% RSLogix 500 project MM2.RSS, saved by version 8.10.00.30 %
PROJECT "UNTITLED"    % processor: Bul.1763 MicroLogix 1100 Series B %

PROGRAM FILES
  LAD 2   4 rungs
  LAD 3 "WATCHDOG"  8 rungs
  LAD 4 "PRODUCT"  8 rungs  % Changes the productcode %

DATA FILES
  O0 OUTPUT  4 elements
  I1 INPUT  6 elements
  S2 STATUS  66 elements
  B3 BINARY  1 elements
  T4 TIMER  3 elements
  C5 COUNTER  1 elements
  R6 CONTROL  1 elements
  N7 INTEGER  3 elements
  F8 FLOAT  100 elements
  ST9   10 elements
  MG13   1 elements
  RIX15   1 elements
  RI16   1 elements

LADDER 2
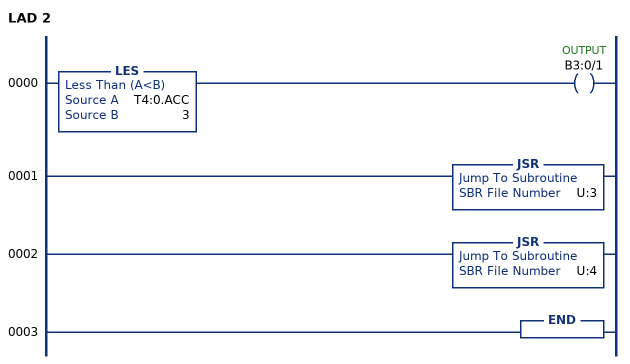
% Rung: 0 %
SOR LES T4:0.ACC 3 OTE B3:0/1 EOR
%   B3:0/1  OUTPUT %
% Rung: 1 %
SOR JSR U:3 EOR
% Rung: 2 %
SOR JSR U:4 EOR
% Rung: 3 %
SOR END EOR

LADDER 3 "WATCHDOG"
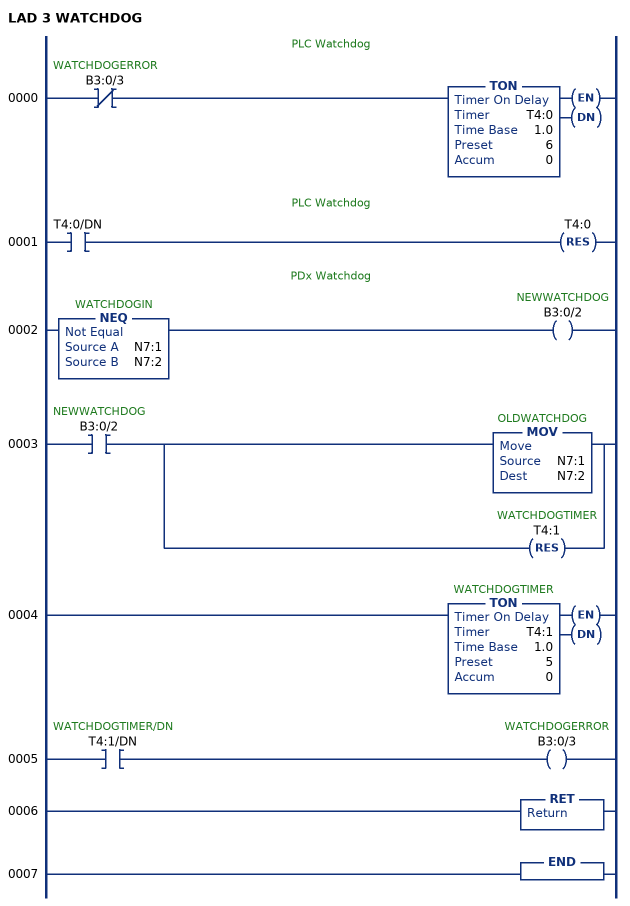
% Rung: 0 %  % edit flag set %
% PLC Watchdog %
SOR XIO B3:0/3 TON T4:0 1.0 6 0 EOR
%   B3:0/3  WATCHDOGERROR %
% Rung: 1 %  % edit flag set %
% PLC Watchdog %
SOR XIC T4:0/DN RES T4:0 EOR
% Rung: 2 %
% PDx Watchdog %
SOR NEQ N7:1 N7:2 OTE B3:0/2 EOR
%   N7:1  WATCHDOGIN %
%   N7:2  OLDWATCHDOG %
%   B3:0/2  NEWWATCHDOG %
% Rung: 3 %
SOR XIC B3:0/2 BST MOV N7:1 N7:2 NXB RES T4:1 BND EOR
%   B3:0/2  NEWWATCHDOG %
%   N7:1  WATCHDOGIN %
%   N7:2  OLDWATCHDOG %
%   T4:1  WATCHDOGTIMER %
% Rung: 4 %
SOR TON T4:1 1.0 5 0 EOR
%   T4:1  WATCHDOGTIMER %
% Rung: 5 %
SOR XIC T4:1/DN OTE B3:0/3 EOR
%   T4:1  WATCHDOGTIMER %
%   B3:0/3  WATCHDOGERROR %
% Rung: 6 %
SOR RET EOR
% Rung: 7 %
SOR END EOR

LADDER 4 "PRODUCT"    % Changes the productcode %
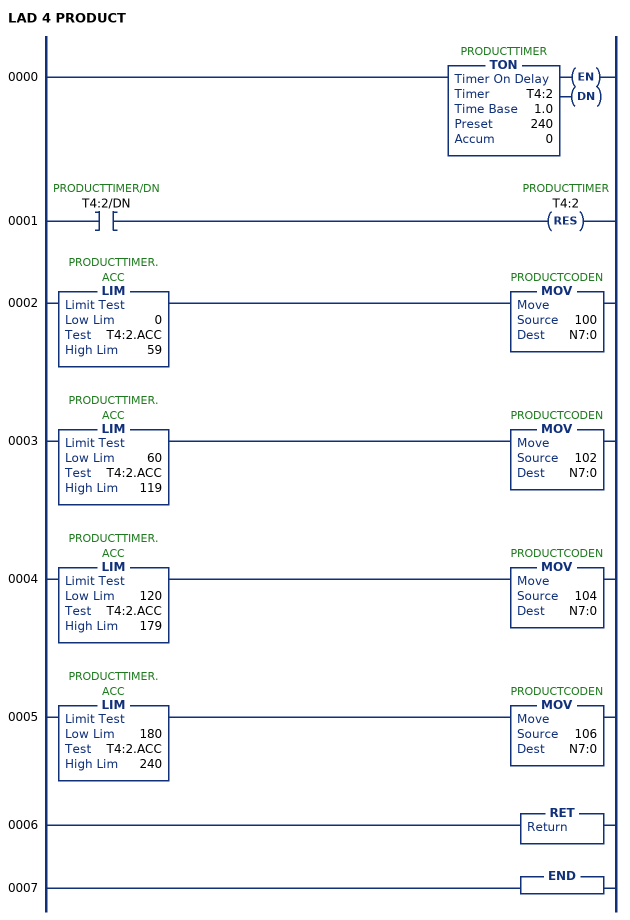
% Rung: 0 %
SOR TON T4:2 1.0 240 0 EOR
%   T4:2  PRODUCTTIMER %
% Rung: 1 %
SOR XIC T4:2/DN RES T4:2 EOR
%   T4:2  PRODUCTTIMER %
% Rung: 2 %
SOR LIM 0 T4:2.ACC 59 MOV 100 N7:0 EOR
%   T4:2  PRODUCTTIMER %
%   N7:0  PRODUCTCODEN %
% Rung: 3 %
SOR LIM 60 T4:2.ACC 119 MOV 102 N7:0 EOR
%   T4:2  PRODUCTTIMER %
%   N7:0  PRODUCTCODEN %
% Rung: 4 %
SOR LIM 120 T4:2.ACC 179 MOV 104 N7:0 EOR
%   T4:2  PRODUCTTIMER %
%   N7:0  PRODUCTCODEN %
% Rung: 5 %
SOR LIM 180 T4:2.ACC 240 MOV 106 N7:0 EOR
%   T4:2  PRODUCTTIMER %
%   N7:0  PRODUCTCODEN %
% Rung: 6 %
SOR RET EOR
% Rung: 7 %
SOR END EOR

OTHER DOCUMENTED ADDRESSES
  B3:0/0  INPUT

DATA TABLE (non-zero values as saved)
DATA B3
% B3:0 % 0X0002
DATA T4
% .PRE .ACC %
% T4:0 % 6 0
% T4:1 % 5 0
% T4:2 % 240 0
DATA C5
% .PRE .ACC %
% C5:0 % 10 0
DATA F8
% F8:0 % 65 0 0 0 0
DATA ST9
% ST9:0 % "3"
% ST9:1 % "FDGDGSFB"
% ST9:3 % "GJGJFGN TRFGHNGD"
